SUBAPPLICATION Ramp6Buttons (* Subapplication Type *)
  (* Standard: 61499-2 *)
  (* Version 1.0, 2026-08-29, franz *)
  PACKAGE MyLib::sys;
  IMPORT isobus::UT::io::Button::ButtonActivationCode::BT_PRESSED_LATCHED;
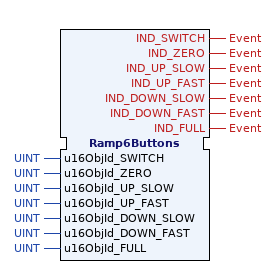
  EVENT_OUTPUT
    IND_SWITCH; (* Kanal-Ein/Aus-Taste gedrueckt (togglet Enable-Zustand) *)
    IND_ZERO; (* Taste '0' gedrueckt (RampLimitFS.ZERO) *)
    IND_UP_SLOW; (* Taste '+' gedrueckt (RampLimitFS.UP_SLOW, ~1%) *)
    IND_UP_FAST; (* Taste '++' gedrueckt (RampLimitFS.UP_FAST, ~10%) *)
    IND_DOWN_SLOW; (* Taste '-' gedrueckt (RampLimitFS.DOWN_SLOW, ~1%) *)
    IND_DOWN_FAST; (* Taste '--' gedrueckt (RampLimitFS.DOWN_FAST, ~10%) *)
    IND_FULL; (* Taste 'F' gedrueckt (RampLimitFS.FULL, 100%) *)
  END_EVENT
  VAR_INPUT
    u16ObjId_SWITCH : UINT;
    u16ObjId_ZERO : UINT;
    u16ObjId_UP_SLOW : UINT;
    u16ObjId_UP_FAST : UINT;
    u16ObjId_DOWN_SLOW : UINT;
    u16ObjId_DOWN_FAST : UINT;
    u16ObjId_FULL : UINT;
  END_VAR
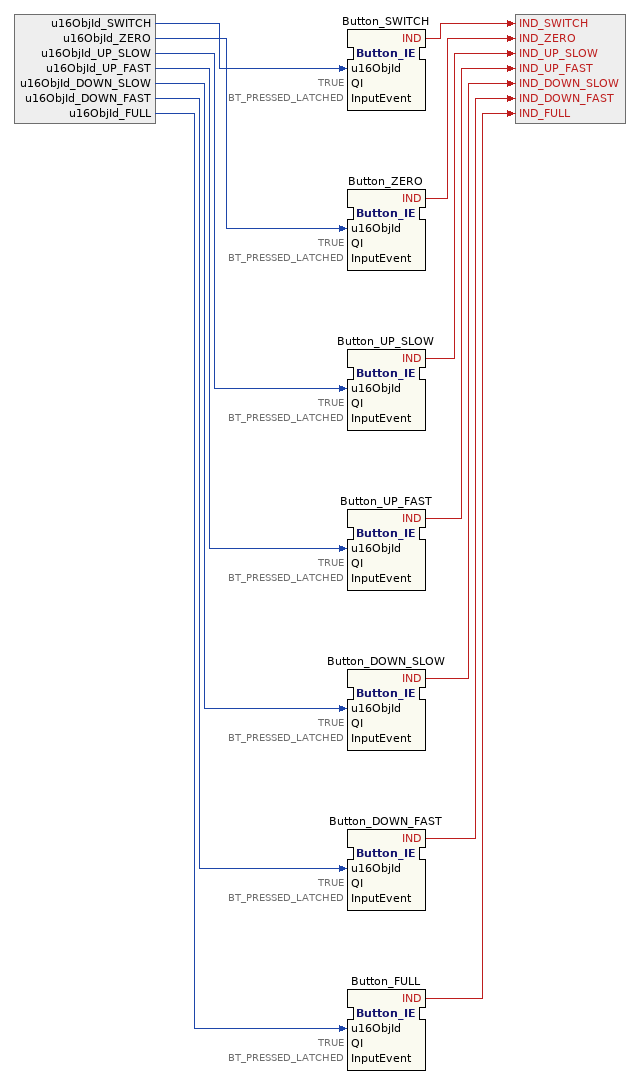
  FBS
    Button_SWITCH : isobus::UT::io::Button::Button_IE(QI := TRUE, InputEvent := BT_PRESSED_LATCHED);
    Button_ZERO : isobus::UT::io::Button::Button_IE(QI := TRUE, InputEvent := BT_PRESSED_LATCHED);
    Button_UP_SLOW : isobus::UT::io::Button::Button_IE(QI := TRUE, InputEvent := BT_PRESSED_LATCHED);
    Button_UP_FAST : isobus::UT::io::Button::Button_IE(QI := TRUE, InputEvent := BT_PRESSED_LATCHED);
    Button_DOWN_SLOW : isobus::UT::io::Button::Button_IE(QI := TRUE, InputEvent := BT_PRESSED_LATCHED);
    Button_DOWN_FAST : isobus::UT::io::Button::Button_IE(QI := TRUE, InputEvent := BT_PRESSED_LATCHED);
    Button_FULL : isobus::UT::io::Button::Button_IE(QI := TRUE, InputEvent := BT_PRESSED_LATCHED);
  END_FBS
  EVENT_CONNECTIONS
    Button_SWITCH.IND TO IND_SWITCH;
    Button_ZERO.IND TO IND_ZERO;
    Button_UP_SLOW.IND TO IND_UP_SLOW;
    Button_UP_FAST.IND TO IND_UP_FAST;
    Button_DOWN_SLOW.IND TO IND_DOWN_SLOW;
    Button_DOWN_FAST.IND TO IND_DOWN_FAST;
    Button_FULL.IND TO IND_FULL;
  END_CONNECTIONS
  DATA_CONNECTIONS
    u16ObjId_SWITCH TO Button_SWITCH.u16ObjId;
    u16ObjId_ZERO TO Button_ZERO.u16ObjId;
    u16ObjId_UP_SLOW TO Button_UP_SLOW.u16ObjId;
    u16ObjId_UP_FAST TO Button_UP_FAST.u16ObjId;
    u16ObjId_DOWN_SLOW TO Button_DOWN_SLOW.u16ObjId;
    u16ObjId_DOWN_FAST TO Button_DOWN_FAST.u16ObjId;
    u16ObjId_FULL TO Button_FULL.u16ObjId;
  END_CONNECTIONS
END_SUBAPPLICATION
